(* Index FB
A. Wallace 2016-9-3

Why doesn't beckhoff have this as a builtin type?

Use this thing to have a simple indexer with rollover.

*)
{attribute 'analysis' := '-2'}
FUNCTION_BLOCK FB_Index
VAR_INPUT
	{attribute 'naming' := 'off'}
	LowerLimit : INT := 1; //Incrementer will rollver over to this value (and initialize to this value)
	ValInc : INT := 1; //Incrementer increments by this value
	UpperLimit	:	INT := 1; //Incrementer will rollover at this value to lower limit
	{attribute 'naming' := 'off'}
END_VAR
VAR_OUTPUT
	
END_VAR
VAR
	nVal	:	INT := LowerLimit; //Internal incrementer value, initialized to LowerLimit
END_VAR

ACTION Dec:
nVal := nVal - ValInc;
IF nVal < LowerLimit THEN nVal := UpperLimit; END_IF
END_ACTION

//Decrement the counter and return new value
METHOD DecVal : INT
VAR_INPUT
END_VAR
Dec();
DecVal := nVal;
END_METHOD

ACTION Inc:
// Dont use this, use ValInc
nVal := nVal + ValInc;
IF nVal >  UpperLimit THEN nVal := LowerLimit; END_IF
END_ACTION

//Increment the counter and return new value
METHOD PUBLIC IncVal : INT
VAR_INPUT
END_VAR
Inc();
IncVal := nVal;
END_METHOD

END_FUNCTION_BLOCK

(* stored: Version 1.1.0.1, ProductVersion 3.1.4022.12
   POU FB_Index: Id {ca8a34e3-bd4f-442e-9caf-17285b4f6fa2}, SpecialFunc None
   Action Dec: Id {b1b81818-0c2b-42cc-90f3-55cd7cad3e87}
   Method DecVal: Id {cf4e17a1-86cd-4a59-ad6f-fc3838ffede5}
   Action Inc: Id {a11e830b-c881-456f-af74-5a750bccfd58}
   Method IncVal: Id {6f28d89a-7191-4dad-8824-c5fe9fb32dd9} *)
